   E6POS P2_G_1_App1Place={X 149.37352,Y -2.09811,Z 1001.61812,A -90,B 0,C 180,S 2,T 51,E1 0,E2 0,E3 0,E4 0,E5 0,E6 0}
   E6POS P2_G_1_App2Place={X 149.37352,Y -2.09821,Z 851.61778,A -90,B 0,C 180,S 2,T 51,E1 0,E2 0,E3 0,E4 0,E5 0,E6 0}
   E6POS P2_G_1_Place={X 49.37367,Y -2.09846,Z 651.61785,A -90,B 0,C 180,S 2,T 51,E1 0,E2 0,E3 0,E4 0,E5 0,E6 0}
   E6POS P2_G_2_App1Place={X 353.37436,Y 585.90188,Z 1001.61812,A -90,B 0,C 180,S 2,T 3,E1 0,E2 0,E3 0,E4 0,E5 0,E6 0}
   E6POS P2_G_2_App2Place={X 353.37434,Y 585.90171,Z 851.61778,A -90,B 0,C 180,S 2,T 3,E1 0,E2 0,E3 0,E4 0,E5 0,E6 0}
   E6POS P2_G_2_Place={X 253.37397,Y 585.90191,Z 651.61785,A -90,B 0,C 180,S 2,T 3,E1 0,E2 0,E3 0,E4 0,E5 0,E6 0}
   E6POS P2_G_3_App1Place={X 162.41236,Y 1308.69058,Z 1001.61812,A -90,B 0,C 180,S 2,T 35,E1 0,E2 0,E3 0,E4 0,E5 0,E6 0}
   E6POS P2_G_3_App2Place={X 162.41236,Y 1308.69069,Z 851.61778,A -90,B 0,C 180,S 2,T 35,E1 0,E2 0,E3 0,E4 0,E5 0,E6 0}
   E6POS P2_G_3_Place={X 49.37239,Y 1173.90187,Z 651.61785,A -90,B 0,C 180,S 2,T 35,E1 0,E2 0,E3 0,E4 0,E5 0,E6 0}
   E6POS P2_G_4_App1Place={X 559.12222,Y -2.23499,Z 1001.61812,A -90,B 0,C -180,S 2,T 19,E1 0,E2 0,E3 0,E4 0,E5 0,E6 0}
   E6POS P2_G_4_App2Place={X 559.12222,Y -2.235,Z 851.61778,A -90,B 0,C 180,S 2,T 19,E1 0,E2 0,E3 0,E4 0,E5 0,E6 0}
   E6POS P2_G_4_Place={X 457.3734,Y -26.09812,Z 651.61785,A -90,B 0,C 180,S 2,T 19,E1 0,E2 0,E3 0,E4 0,E5 0,E6 0}
   E6POS P2_G_5_App1Place={X 566.4018,Y 1306.30275,Z 1001.61812,A -90,B 0,C -180,S 2,T 3,E1 0,E2 0,E3 0,E4 0,E5 0,E6 0}
   E6POS P2_G_5_App2Place={X 566.4018,Y 1306.30279,Z 851.61778,A -90,B 0,C 180,S 2,T 3,E1 0,E2 0,E3 0,E4 0,E5 0,E6 0}
   E6POS P2_G_5_Place={X 343.37167,Y 1197.90666,Z 651.61785,A -90,B 0,C 180,S 2,T 3,E1 0,E2 0,E3 0,E4 0,E5 0,E6 0}
   E6POS P2_G_6_App1Place={X 770.4018,Y 1306.30275,Z 1001.61812,A -90,B 0,C -180,S 2,T 3,E1 0,E2 0,E3 0,E4 0,E5 0,E6 0}
   E6POS P2_G_6_App2Place={X 770.4018,Y 1306.30279,Z 851.61778,A -90,B 0,C 180,S 2,T 3,E1 0,E2 0,E3 0,E4 0,E5 0,E6 0}
   E6POS P2_G_6_Place={X 547.37167,Y 1197.90666,Z 651.61785,A -90,B 0,C 180,S 2,T 3,E1 0,E2 0,E3 0,E4 0,E5 0,E6 0}
   E6POS P2_G_7_App1Place={X 853.12026,Y 609.77279,Z 1001.61812,A -89.99997,B 0,C -180,S 2,T 3,E1 0,E2 0,E3 0,E4 0,E5 0,E6 0}
   E6POS P2_G_7_App2Place={X 853.12035,Y 609.77308,Z 851.61778,A -89.99997,B 0,C 180,S 2,T 3,E1 0,E2 0,E3 0,E4 0,E5 0,E6 0}
   E6POS P2_G_7_Place={X 751.37887,Y 612.61574,Z 651.61785,A -89.99997,B 0,C 180,S 2,T 3,E1 0,E2 0,E3 0,E4 0,E5 0,E6 0}
   E6POS P2_G_8_App1Place={X 753.12073,Y 609.77254,Z 1001.61812,A -90,B 0,C 180,S 2,T 3,E1 0,E2 0,E3 0,E4 0,E5 0,E6 0}
   E6POS P2_G_8_App2Place={X 753.12006,Y 654.77255,Z 851.61778,A -89.99997,B 0,C 180,S 2,T 3,E1 0,E2 0,E3 0,E4 0,E5 0,E6 0}
   E6POS P2_G_8_Place={X 753.12003,Y 654.77244,Z 651.61785,A -89.99997,B 0,C 180,S 2,T 3,E1 0,E2 0,E3 0,E4 0,E5 0,E6 0}
   E6POS P2_G_9_App1Place={X 753.12006,Y 654.77255,Z 1001.61812,A -89.99997,B 0,C 180,S 2,T 3,E1 0,E2 0,E3 0,E4 0,E5 0,E6 0}
   E6POS P2_G_9_App2Place={X 753.12053,Y 699.77216,Z 851.61778,A -90,B 0,C 180,S 2,T 3,E1 0,E2 0,E3 0,E4 0,E5 0,E6 0}
   E6POS P2_G_9_Place={X 753.12063,Y 699.77251,Z 651.61785,A -90,B 0,C 180,S 2,T 3,E1 0,E2 0,E3 0,E4 0,E5 0,E6 0}
   E6POS P2_G_10_App1Place={X 753.12053,Y 699.77216,Z 1001.61812,A -90,B 0,C 180,S 2,T 3,E1 0,E2 0,E3 0,E4 0,E5 0,E6 0}
   E6POS P2_G_10_App2Place={X 753.12058,Y 744.7725,Z 851.61778,A -90,B 0,C 180,S 2,T 3,E1 0,E2 0,E3 0,E4 0,E5 0,E6 0}
   E6POS P2_G_10_Place={X 753.12059,Y 744.77255,Z 651.61785,A -90,B 0,C 180,S 2,T 3,E1 0,E2 0,E3 0,E4 0,E5 0,E6 0}
   E6POS P2_G_11_App1Place={X 753.12058,Y 744.7725,Z 1001.61812,A -90,B 0,C 180,S 2,T 3,E1 0,E2 0,E3 0,E4 0,E5 0,E6 0}
   E6POS P2_G_11_App2Place={X 753.12054,Y 789.7722,Z 851.61778,A -90,B 0,C 180,S 2,T 3,E1 0,E2 0,E3 0,E4 0,E5 0,E6 0}
   E6POS P2_G_11_Place={X 753.12064,Y 789.7726,Z 651.61785,A -90,B 0,C 180,S 2,T 3,E1 0,E2 0,E3 0,E4 0,E5 0,E6 0}
   E6POS P2_G_12_App1Place={X 443.37199,Y 585.90705,Z 1001.61812,A -90,B 0,C -180,S 2,T 3,E1 0,E2 0,E3 0,E4 0,E5 0,E6 0}
   E6POS P2_G_12_App2Place={X 443.37195,Y 585.90667,Z 851.61778,A -90,B 0,C 180,S 2,T 3,E1 0,E2 0,E3 0,E4 0,E5 0,E6 0}
   E6POS P2_G_12_Place={X 343.37181,Y 585.90688,Z 651.61785,A -90,B 0,C 180,S 2,T 3,E1 0,E2 0,E3 0,E4 0,E5 0,E6 0}
   E6POS P2_G_13_App1Place={X 647.37185,Y -2.09309,Z 1001.61812,A -90,B 0,C -180,S 2,T 3,E1 0,E2 0,E3 0,E4 0,E5 0,E6 0}
   E6POS P2_G_13_App2Place={X 647.37173,Y -2.09348,Z 851.61778,A -90,B 0,C 180,S 2,T 3,E1 0,E2 0,E3 0,E4 0,E5 0,E6 0}
   E6POS P2_G_13_Place={X 547.37181,Y -2.0932,Z 651.61785,A -90,B 0,C 180,S 2,T 19,E1 0,E2 0,E3 0,E4 0,E5 0,E6 0}
   E6POS P2_G_14_App1Place={X 393.37089,Y 1223.90695,Z 1001.61812,A -90,B 0,C 180,S 2,T 3,E1 0,E2 0,E3 0,E4 0,E5 0,E6 0}
   E6POS P2_G_14_App2Place={X 393.37089,Y 1223.90695,Z 851.61778,A -90,B 0,C 180,S 2,T 3,E1 0,E2 0,E3 0,E4 0,E5 0,E6 0}
   E6POS P2_G_14_Place={X 343.37089,Y 1173.90695,Z 651.61785,A -90,B 0,C 180,S 2,T 3,E1 0,E2 0,E3 0,E4 0,E5 0,E6 0}
   E6POS P2_G_15_App1Place={X 853.11933,Y -26.09364,Z 1001.61812,A -90,B 0,C -180,S 2,T 3,E1 0,E2 0,E3 0,E4 0,E5 0,E6 0}
   E6POS P2_G_15_App2Place={X 853.11941,Y -26.09348,Z 851.61778,A -90,B 0,C 180,S 2,T 3,E1 0,E2 0,E3 0,E4 0,E5 0,E6 0}
   E6POS P2_G_15_Place={X 751.37143,Y -26.09385,Z 651.61785,A -90,B 0,C 180,S 2,T 19,E1 0,E2 0,E3 0,E4 0,E5 0,E6 0}
   E6POS P2_G_16_App1Place={X 737.36387,Y 1297.90653,Z 1001.61812,A -90,B 0,C -180,S 2,T 3,E1 0,E2 0,E3 0,E4 0,E5 0,E6 0}
   E6POS P2_G_16_App2Place={X 737.36384,Y 1297.90637,Z 851.61778,A -90,B 0,C 180,S 2,T 3,E1 0,E2 0,E3 0,E4 0,E5 0,E6 0}
   E6POS P2_G_16_Place={X 637.37555,Y 1197.90665,Z 651.61785,A -90,B 0,C 180,S 2,T 3,E1 0,E2 0,E3 0,E4 0,E5 0,E6 0}
   E6POS P2_G_17_App1Place={X 941.36387,Y 1297.90653,Z 1001.61812,A -90,B 0,C -180,S 2,T 3,E1 0,E2 0,E3 0,E4 0,E5 0,E6 0}
   E6POS P2_G_17_App2Place={X 941.36384,Y 1297.90637,Z 851.61778,A -90,B 0,C -180,S 2,T 3,E1 0,E2 0,E3 0,E4 0,E5 0,E6 0}
   E6POS P2_G_17_Place={X 841.37555,Y 1197.90665,Z 651.61785,A -90,B 0,C -180,S 2,T 3,E1 0,E2 0,E3 0,E4 0,E5 0,E6 0}
   E6POS P2_G_18_App1Place={X 75.37306,Y 583.87483,Z 1001.61812,A 90,B 0,C -180,S 2,T 35,E1 0,E2 0,E3 0,E4 0,E5 0,E6 0}
   E6POS P2_G_18_App2Place={X 75.37307,Y 583.87481,Z 851.61778,A 90,B 0,C 180,S 2,T 35,E1 0,E2 0,E3 0,E4 0,E5 0,E6 0}
   E6POS P2_G_18_Place={X 220.62117,Y 583.87476,Z 651.61785,A 90,B 0,C 180,S 2,T 35,E1 0,E2 0,E3 0,E4 0,E5 0,E6 0}
   E6POS P2_G_19_App1Place={X 220.62116,Y 583.87476,Z 1001.61812,A 90,B 0,C 180,S 2,T 35,E1 0,E2 0,E3 0,E4 0,E5 0,E6 0}
   E6POS P2_G_19_App2Place={X 220.62116,Y 538.87476,Z 851.61778,A 90,B 0,C 180,S 2,T 35,E1 0,E2 0,E3 0,E4 0,E5 0,E6 0}
   E6POS P2_G_19_Place={X 220.62116,Y 538.87476,Z 651.61785,A 90,B 0,C 180,S 2,T 35,E1 0,E2 0,E3 0,E4 0,E5 0,E6 0}
   E6POS P2_G_20_App1Place={X 220.62116,Y 538.87476,Z 1001.61812,A 90,B 0,C 180,S 2,T 35,E1 0,E2 0,E3 0,E4 0,E5 0,E6 0}
   E6POS P2_G_20_App2Place={X 220.62116,Y 493.87476,Z 851.61778,A 90,B 0,C 180,S 2,T 35,E1 0,E2 0,E3 0,E4 0,E5 0,E6 0}
   E6POS P2_G_20_Place={X 220.62116,Y 493.87476,Z 651.61785,A 90,B 0,C 180,S 2,T 35,E1 0,E2 0,E3 0,E4 0,E5 0,E6 0}
   E6POS P2_G_21_App1Place={X 220.62116,Y 493.87476,Z 1001.61812,A 90,B 0,C 180,S 2,T 35,E1 0,E2 0,E3 0,E4 0,E5 0,E6 0}
   E6POS P2_G_21_App2Place={X 220.62116,Y 448.87476,Z 851.61778,A 90,B 0,C 180,S 2,T 35,E1 0,E2 0,E3 0,E4 0,E5 0,E6 0}
   E6POS P2_G_21_Place={X 220.62116,Y 448.87476,Z 651.61785,A 90,B 0,C 180,S 2,T 35,E1 0,E2 0,E3 0,E4 0,E5 0,E6 0}
   E6POS P2_G_22_App1Place={X 220.62116,Y 448.87476,Z 1001.61812,A 90,B 0,C 180,S 2,T 35,E1 0,E2 0,E3 0,E4 0,E5 0,E6 0}
   E6POS P2_G_22_App2Place={X 220.62116,Y 403.87476,Z 851.61778,A 90,B 0,C 180,S 2,T 35,E1 0,E2 0,E3 0,E4 0,E5 0,E6 0}
   E6POS P2_G_22_Place={X 220.62116,Y 403.87476,Z 651.61785,A 90,B 0,C 180,S 2,T 35,E1 0,E2 0,E3 0,E4 0,E5 0,E6 0}

   ;ENDFOLD
   ;FOLD  MosaicoI_Pallet2

   E6POS P2_I_1_App1Place={X 246.53077,Y 662.7024,Z 986.30178,A -90,B 0,C 180,S 2,T 3,E1 0,E2 0,E3 0,E4 0,E5 0,E6 0}
   E6POS P2_I_1_App2Place={X 246.53091,Y 662.7025,Z 836.30179,A -90,B 0,C 180,S 2,T 3,E1 0,E2 0,E3 0,E4 0,E5 0,E6 0}
   E6POS P2_I_1_Place={X 120.2419,Y 563.31321,Z 652.09239,A -90,B 0,C 180,S 2,T 35,E1 0,E2 0,E3 0,E4 0,E5 0,E6 0}
   E6POS P2_I_2_App1Place={X 120.24188,Y 563.31279,Z 986.30178,A -90,B 0,C 180,S 2,T 35,E1 0,E2 0,E3 0,E4 0,E5 0,E6 0}
   E6POS P2_I_2_App2Place={X 120.24229,Y 624.31271,Z 836.30179,A -90,B 0,C 180,S 2,T 35,E1 0,E2 0,E3 0,E4 0,E5 0,E6 0}
   E6POS P2_I_2_Place={X 120.24227,Y 624.3123,Z 652.09239,A -90,B 0,C 180,S 2,T 35,E1 0,E2 0,E3 0,E4 0,E5 0,E6 0}
   E6POS P2_I_3_App1Place={X 120.24229,Y 624.31271,Z 986.30178,A -90,B 0,C 180,S 2,T 35,E1 0,E2 0,E3 0,E4 0,E5 0,E6 0}
   E6POS P2_I_3_App2Place={X 120.24194,Y 685.31244,Z 836.30179,A -90,B 0,C 180,S 2,T 35,E1 0,E2 0,E3 0,E4 0,E5 0,E6 0}
   E6POS P2_I_3_Place={X 120.24196,Y 685.31272,Z 652.09239,A -90,B 0,C 180,S 2,T 35,E1 0,E2 0,E3 0,E4 0,E5 0,E6 0}
   E6POS P2_I_4_App1Place={X 584.7347,Y 593.50005,Z 986.30178,A 90,B 0,C 180,S 2,T 35,E1 0,E2 0,E3 0,E4 0,E5 0,E6 0}
   E6POS P2_I_4_App2Place={X 584.73528,Y 593.49987,Z 836.30179,A 90,B 0,C 180,S 2,T 35,E1 0,E2 0,E3 0,E4 0,E5 0,E6 0}
   E6POS P2_I_4_Place={X 484.73518,Y 593.50008,Z 652.09239,A 90,B 0,C 180,S 2,T 35,E1 0,E2 0,E3 0,E4 0,E5 0,E6 0}
   E6POS P2_I_5_App1Place={X 942.73548,Y 593.50065,Z 986.30178,A 90,B 0,C 180,S 2,T 35,E1 0,E2 0,E3 0,E4 0,E5 0,E6 0}
   E6POS P2_I_5_App2Place={X 942.73575,Y 593.50015,Z 836.30179,A 90,B 0,C 180,S 2,T 35,E1 0,E2 0,E3 0,E4 0,E5 0,E6 0}
   E6POS P2_I_5_Place={X 842.73579,Y 593.50005,Z 652.09239,A 90,B 0,C 180,S 2,T 35,E1 0,E2 0,E3 0,E4 0,E5 0,E6 0}
   E6POS P2_I_6_App1Place={X 413.73426,Y 594.42093,Z 986.30178,A 90,B 0,C 180,S 2,T 35,E1 0,E2 0,E3 0,E4 0,E5 0,E6 0}
   E6POS P2_I_6_App2Place={X 413.73463,Y 594.42083,Z 836.30179,A 90,B 0,C 180,S 2,T 35,E1 0,E2 0,E3 0,E4 0,E5 0,E6 0}
   E6POS P2_I_6_Place={X 313.73464,Y 594.42082,Z 652.09239,A 90,B 0,C 180,S 2,T 35,E1 0,E2 0,E3 0,E4 0,E5 0,E6 0}
   E6POS P2_I_7_App1Place={X 771.7338,Y 594.4204,Z 986.30178,A 90,B 0,C 180,S 2,T 35,E1 0,E2 0,E3 0,E4 0,E5 0,E6 0}
   E6POS P2_I_7_App2Place={X 771.73418,Y 594.4208,Z 836.30179,A 90,B 0,C 180,S 2,T 35,E1 0,E2 0,E3 0,E4 0,E5 0,E6 0}
   E6POS P2_I_7_Place={X 671.73443,Y 594.42068,Z 652.09239,A 90,B 0,C 180,S 2,T 35,E1 0,E2 0,E3 0,E4 0,E5 0,E6 0}
   E6POS P2_I_8_App1Place={X 936.24205,Y 563.31282,Z 986.30178,A -90,B 0,C 180,S 2,T 3,E1 0,E2 0,E3 0,E4 0,E5 0,E6 0}
   E6POS P2_I_8_App2Place={X 936.24164,Y 563.31281,Z 836.30179,A -90,B 0,C 180,S 2,T 3,E1 0,E2 0,E3 0,E4 0,E5 0,E6 0}
   E6POS P2_I_8_Place={X 836.24218,Y 563.31266,Z 652.09239,A -90,B 0,C 180,S 2,T 3,E1 0,E2 0,E3 0,E4 0,E5 0,E6 0}
   E6POS P2_I_9_App1Place={X 836.24219,Y 563.31262,Z 986.30178,A -90,B 0,C 180,S 2,T 3,E1 0,E2 0,E3 0,E4 0,E5 0,E6 0}
   E6POS P2_I_9_App2Place={X 836.24173,Y 624.31272,Z 836.30179,A -90,B 0,C 180,S 2,T 3,E1 0,E2 0,E3 0,E4 0,E5 0,E6 0}
   E6POS P2_I_9_Place={X 836.24181,Y 624.31245,Z 652.09239,A -90,B 0,C 180,S 2,T 3,E1 0,E2 0,E3 0,E4 0,E5 0,E6 0}
   E6POS P2_I_10_App1Place={X 836.24173,Y 624.31272,Z 986.30178,A -90,B 0,C 180,S 2,T 3,E1 0,E2 0,E3 0,E4 0,E5 0,E6 0}
   E6POS P2_I_10_App2Place={X 836.24228,Y 685.31292,Z 836.30179,A -90,B 0,C 180,S 2,T 3,E1 0,E2 0,E3 0,E4 0,E5 0,E6 0}
   E6POS P2_I_10_Place={X 836.24232,Y 685.3128,Z 652.09239,A -90,B 0,C 180,S 2,T 3,E1 0,E2 0,E3 0,E4 0,E5 0,E6 0}

   ;ENDFOLD
   ;FOLD  MosaicoJ_Pallet2

   E6POS P2_J_1_App1Place={X 205.12202,Y 673.01054,Z 986.30252,A 90,B 0,C 180,S 2,T 35,E1 0,E2 0,E3 0,E4 0,E5 0,E6 0}
   E6POS P2_J_1_App2Place={X 205.12222,Y 673.01047,Z 786.30223,A 90,B 0,C 180,S 2,T 35,E1 0,E2 0,E3 0,E4 0,E5 0,E6 0}
   E6POS P2_J_1_Place={X 83.2071,Y 563.55362,Z 666.3006,A 90,B 0,C 180,S 2,T 35,E1 0,E2 0,E3 0,E4 0,E5 0,E6 0}
   E6POS P2_J_2_App1Place={X 996.70818,Y 190.44821,Z 986.30252,A -180,B 0,C -180,S 2,T 35,E1 0,E2 0,E3 0,E4 0,E5 0,E6 0}
   E6POS P2_J_2_App2Place={X 996.70793,Y 190.44835,Z 786.30223,A -180,B 0,C 180,S 2,T 35,E1 0,E2 0,E3 0,E4 0,E5 0,E6 0}
   E6POS P2_J_2_Place={X 896.70882,Y 90.44837,Z 666.3006,A -180,B 0,C -180,S 2,T 51,E1 0,E2 0,E3 0,E4 0,E5 0,E6 0}
   E6POS P2_J_3_App1Place={X 996.70874,Y 479.44951,Z 986.30252,A -180,B 0,C 180,S 2,T 35,E1 0,E2 0,E3 0,E4 0,E5 0,E6 0}
   E6POS P2_J_3_App2Place={X 996.70888,Y 479.44931,Z 786.30223,A -180,B 0,C 180,S 2,T 35,E1 0,E2 0,E3 0,E4 0,E5 0,E6 0}
   E6POS P2_J_3_Place={X 896.7079,Y 379.44856,Z 666.3006,A -180,B 0,C 180,S 2,T 35,E1 0,E2 0,E3 0,E4 0,E5 0,E6 0}
   E6POS P2_J_4_App1Place={X 996.70922,Y 768.44904,Z 986.30252,A -180,B 0,C 180,S 2,T 35,E1 0,E2 0,E3 0,E4 0,E5 0,E6 0}
   E6POS P2_J_4_App2Place={X 996.70882,Y 768.44907,Z 786.30223,A -180,B 0,C 180,S 2,T 35,E1 0,E2 0,E3 0,E4 0,E5 0,E6 0}
   E6POS P2_J_4_Place={X 896.708,Y 668.44849,Z 666.3006,A -180,B 0,C 180,S 2,T 35,E1 0,E2 0,E3 0,E4 0,E5 0,E6 0}
   E6POS P2_J_5_App1Place={X 996.70917,Y 1057.44893,Z 986.30252,A -180,B 0,C 180,S 2,T 35,E1 0,E2 0,E3 0,E4 0,E5 0,E6 0}
   E6POS P2_J_5_App2Place={X 996.70891,Y 1057.44895,Z 786.30223,A -180,B 0,C -180,S 2,T 35,E1 0,E2 0,E3 0,E4 0,E5 0,E6 0}
   E6POS P2_J_5_Place={X 896.7083,Y 957.44855,Z 666.3006,A -180,B 0,C 180,S 2,T 35,E1 0,E2 0,E3 0,E4 0,E5 0,E6 0}
   E6POS P2_J_6_App1Place={X 624.70927,Y 190.44867,Z 986.30252,A -180,B 0,C 180,S 2,T 35,E1 0,E2 0,E3 0,E4 0,E5 0,E6 0}
   E6POS P2_J_6_App2Place={X 624.70884,Y 190.44885,Z 786.30223,A -180,B 0,C -180,S 2,T 35,E1 0,E2 0,E3 0,E4 0,E5 0,E6 0}
   E6POS P2_J_6_Place={X 624.70888,Y 90.44835,Z 666.3006,A -180,B 0,C 180,S 2,T 35,E1 0,E2 0,E3 0,E4 0,E5 0,E6 0}
   E6POS P2_J_7_App1Place={X 624.70769,Y 479.44883,Z 986.30252,A -180,B 0,C 180,S 2,T 35,E1 0,E2 0,E3 0,E4 0,E5 0,E6 0}
   E6POS P2_J_7_App2Place={X 624.70799,Y 479.4485,Z 786.30223,A -180,B 0,C 180,S 2,T 35,E1 0,E2 0,E3 0,E4 0,E5 0,E6 0}
   E6POS P2_J_7_Place={X 624.70786,Y 379.44821,Z 666.3006,A -180,B 0,C -180,S 2,T 35,E1 0,E2 0,E3 0,E4 0,E5 0,E6 0}
   E6POS P2_J_8_App1Place={X 624.70801,Y 768.44835,Z 986.30252,A -180,B 0,C 180,S 2,T 35,E1 0,E2 0,E3 0,E4 0,E5 0,E6 0}
   E6POS P2_J_8_App2Place={X 624.70825,Y 768.44844,Z 786.30223,A -180,B 0,C 180,S 2,T 35,E1 0,E2 0,E3 0,E4 0,E5 0,E6 0}
   E6POS P2_J_8_Place={X 624.70846,Y 668.44829,Z 666.3006,A -180,B 0,C -180,S 2,T 35,E1 0,E2 0,E3 0,E4 0,E5 0,E6 0}
   E6POS P2_J_9_App1Place={X 624.70855,Y 1057.44886,Z 986.30252,A -180,B 0,C -180,S 2,T 35,E1 0,E2 0,E3 0,E4 0,E5 0,E6 0}
   E6POS P2_J_9_App2Place={X 624.70849,Y 1057.44878,Z 786.30223,A -180,B 0,C -180,S 2,T 35,E1 0,E2 0,E3 0,E4 0,E5 0,E6 0}
   E6POS P2_J_9_Place={X 624.7086,Y 957.44847,Z 666.3006,A -180,B 0,C 180,S 2,T 35,E1 0,E2 0,E3 0,E4 0,E5 0,E6 0}
   E6POS P2_J_10_App1Place={X 867.21049,Y 562.58511,Z 986.30252,A 90,B 0,C 180,S 2,T 35,E1 0,E2 0,E3 0,E4 0,E5 0,E6 0}
   E6POS P2_J_10_App2Place={X 867.21029,Y 562.58552,Z 786.30223,A 90,B 0,C 180,S 2,T 35,E1 0,E2 0,E3 0,E4 0,E5 0,E6 0}
   E6POS P2_J_10_Place={X 767.21058,Y 562.5858,Z 666.3006,A 90,B 0,C 180,S 2,T 35,E1 0,E2 0,E3 0,E4 0,E5 0,E6 0}

   ;ENDFOLD
   ;FOLD  MosaicoK_Pallet2

   E6POS P2_K_1_App1Place={X 965.18951,Y 160.47376,Z 1002.77257,A -180,B 0,C 180,S 2,T 35,E1 0,E2 0,E3 0,E4 0,E5 0,E6 0}
   E6POS P2_K_1_App2Place={X 965.18946,Y 160.47317,Z 802.77226,A -180,B 0,C 180,S 2,T 35,E1 0,E2 0,E3 0,E4 0,E5 0,E6 0}
   E6POS P2_K_1_Place={X 965.18981,Y 60.47307,Z 652.77183,A -180,B 0,C -180,S 2,T 51,E1 0,E2 0,E3 0,E4 0,E5 0,E6 0}
   E6POS P2_K_2_App1Place={X 289.34869,Y 416.70488,Z 1002.77257,A -180,B 0,C 180,S 2,T 35,E1 0,E2 0,E3 0,E4 0,E5 0,E6 0}
   E6POS P2_K_2_App2Place={X 289.34829,Y 416.70443,Z 802.77226,A -180,B 0,C -180,S 2,T 35,E1 0,E2 0,E3 0,E4 0,E5 0,E6 0}
   E6POS P2_K_2_Place={X 289.34787,Y 316.70418,Z 652.77183,A -180,B 0,C -180,S 2,T 51,E1 0,E2 0,E3 0,E4 0,E5 0,E6 0}
   E6POS P2_K_3_App1Place={X 709.18337,Y 836.49354,Z 1002.77257,A -180,B 0,C 180,S 2,T 35,E1 0,E2 0,E3 0,E4 0,E5 0,E6 0}
   E6POS P2_K_3_App2Place={X 709.18357,Y 836.4934,Z 802.77226,A -180,B 0,C 180,S 2,T 35,E1 0,E2 0,E3 0,E4 0,E5 0,E6 0}
   E6POS P2_K_3_Place={X 709.18379,Y 736.49338,Z 652.77183,A -180,B 0,C -180,S 2,T 35,E1 0,E2 0,E3 0,E4 0,E5 0,E6 0}
   E6POS P2_K_4_App1Place={X 33.34909,Y 1092.70494,Z 1002.77257,A -180,B 0,C -180,S 2,T 35,E1 0,E2 0,E3 0,E4 0,E5 0,E6 0}
   E6POS P2_K_4_App2Place={X 33.34872,Y 1092.70456,Z 802.77226,A -180,B 0,C -180,S 2,T 35,E1 0,E2 0,E3 0,E4 0,E5 0,E6 0}
   E6POS P2_K_4_Place={X 33.34906,Y 992.70434,Z 652.77183,A -180,B 0,C 180,S 2,T 35,E1 0,E2 0,E3 0,E4 0,E5 0,E6 0}
   E6POS P2_K_5_App1Place={X 135.86643,Y -91.91437,Z 1002.77257,A 90,B 0,C 180,S 2,T 51,E1 0,E2 0,E3 0,E4 0,E5 0,E6 0}
   E6POS P2_K_5_App2Place={X 135.86633,Y -91.91463,Z 802.77226,A 90,B 0,C 180,S 2,T 51,E1 0,E2 0,E3 0,E4 0,E5 0,E6 0}
   E6POS P2_K_5_Place={X 230.11027,Y 4.30843,Z 652.77183,A 90,B 0,C 180,S 2,T 51,E1 0,E2 0,E3 0,E4 0,E5 0,E6 0}
   E6POS P2_K_6_App1Place={X 867.49583,Y 1243.09331,Z 1002.77257,A -90.00003,B 0,C 180,S 2,T 3,E1 0,E2 0,E3 0,E4 0,E5 0,E6 0}
   E6POS P2_K_6_App2Place={X 867.4955,Y 1243.0937,Z 802.77226,A -90.00001,B 0,C 180,S 2,T 3,E1 0,E2 0,E3 0,E4 0,E5 0,E6 0}
   E6POS P2_K_6_Place={X 767.4955,Y 1193.0937,Z 652.77183,A -90.00001,B 0,C 180,S 2,T 3,E1 0,E2 0,E3 0,E4 0,E5 0,E6 0}
   E6POS P2_K_7_App1Place={X 709.18372,Y 160.49371,Z 1002.77257,A -180,B 0,C 180,S 2,T 35,E1 0,E2 0,E3 0,E4 0,E5 0,E6 0}
   E6POS P2_K_7_App2Place={X 709.18356,Y 160.49366,Z 802.77226,A -180,B 0,C 180,S 2,T 35,E1 0,E2 0,E3 0,E4 0,E5 0,E6 0}
   E6POS P2_K_7_Place={X 709.18265,Y 60.49314,Z 652.77183,A -180,B 0,C 180,S 2,T 35,E1 0,E2 0,E3 0,E4 0,E5 0,E6 0}
   E6POS P2_K_8_App1Place={X 33.34874,Y 416.70446,Z 1002.77257,A -180,B 0,C 180,S 2,T 35,E1 0,E2 0,E3 0,E4 0,E5 0,E6 0}
   E6POS P2_K_8_App2Place={X 33.34863,Y 416.70468,Z 802.77226,A -180,B 0,C -180,S 2,T 35,E1 0,E2 0,E3 0,E4 0,E5 0,E6 0}
   E6POS P2_K_8_Place={X 33.3492,Y 316.7046,Z 652.77183,A -180,B 0,C -180,S 2,T 35,E1 0,E2 0,E3 0,E4 0,E5 0,E6 0}
   E6POS P2_K_9_App1Place={X 965.18407,Y 836.49236,Z 1002.77257,A -180,B 0,C 180,S 2,T 35,E1 0,E2 0,E3 0,E4 0,E5 0,E6 0}
   E6POS P2_K_9_App2Place={X 965.18406,Y 836.49238,Z 802.77226,A -180,B 0,C 180,S 2,T 35,E1 0,E2 0,E3 0,E4 0,E5 0,E6 0}
   E6POS P2_K_9_Place={X 965.18419,Y 736.49329,Z 652.77183,A -180,B 0,C 180,S 2,T 35,E1 0,E2 0,E3 0,E4 0,E5 0,E6 0}
   E6POS P2_K_10_App1Place={X 289.34853,Y 1092.70485,Z 1002.77257,A -180,B 0,C 180,S 2,T 35,E1 0,E2 0,E3 0,E4 0,E5 0,E6 0}
   E6POS P2_K_10_App2Place={X 289.34898,Y 1092.70437,Z 802.77226,A -180,B 0,C 180,S 2,T 35,E1 0,E2 0,E3 0,E4 0,E5 0,E6 0}
   E6POS P2_K_10_Place={X 289.34887,Y 992.70441,Z 652.77183,A -180,B 0,C -180,S 2,T 35,E1 0,E2 0,E3 0,E4 0,E5 0,E6 0}
   E6POS P2_K_11_App1Place={X 132.98721,Y 1243.0855,Z 1002.77257,A -90,B 0,C 180,S 2,T 35,E1 0,E2 0,E3 0,E4 0,E5 0,E6 0}
   E6POS P2_K_11_App2Place={X 132.98733,Y 1243.08625,Z 802.77226,A -90,B 0,C 180,S 2,T 35,E1 0,E2 0,E3 0,E4 0,E5 0,E6 0}
   E6POS P2_K_11_Place={X 232.98733,Y 1193.08625,Z 652.77183,A -90,B 0,C 180,S 2,T 3,E1 0,E2 0,E3 0,E4 0,E5 0,E6 0}
   E6POS P2_K_12_App1Place={X 864.59574,Y -45.68689,Z 1002.77257,A 90,B 0,C 180,S 2,T 35,E1 0,E2 0,E3 0,E4 0,E5 0,E6 0}
   E6POS P2_K_12_App2Place={X 864.59587,Y -45.68653,Z 802.77226,A 90,B 0,C 180,S 2,T 35,E1 0,E2 0,E3 0,E4 0,E5 0,E6 0}
   E6POS P2_K_12_Place={X 764.59587,Y 4.31347,Z 652.77183,A 90,B 0,C 180,S 2,T 51,E1 0,E2 0,E3 0,E4 0,E5 0,E6 0}

   ;ENDFOLD
   ;FOLD  MosaicoL_Pallet2

   E6POS P2_L_1_App1Place={X 168.06418,Y 598.29338,Z 1070.17203,A -89.99997,B 0,C -180,S 2,T 35,E1 0,E2 0,E3 0,E4 0,E5 0,E6 0}
   E6POS P2_L_1_App2Place={X 168.06418,Y 598.29353,Z 870.17216,A -89.99997,B 0,C 180,S 2,T 35,E1 0,E2 0,E3 0,E4 0,E5 0,E6 0}
   E6POS P2_L_1_Place={X 68.06526,Y 598.29341,Z 670.17152,A -90,B 0,C 180,S 2,T 35,E1 0,E2 0,E3 0,E4 0,E5 0,E6 0}
   E6POS P2_L_2_App1Place={X 432.06392,Y 598.29328,Z 1070.17203,A -89.99997,B 0,C -180,S 2,T 3,E1 0,E2 0,E3 0,E4 0,E5 0,E6 0}
   E6POS P2_L_2_App2Place={X 432.06389,Y 598.29299,Z 870.17216,A -89.99997,B 0,C 180,S 2,T 3,E1 0,E2 0,E3 0,E4 0,E5 0,E6 0}
   E6POS P2_L_2_Place={X 332.06426,Y 598.2932,Z 670.17152,A -89.99997,B 0,C 180,S 2,T 3,E1 0,E2 0,E3 0,E4 0,E5 0,E6 0}
   E6POS P2_L_3_App1Place={X 696.09642,Y 672.2385,Z 1070.17203,A -90,B 0,C -180,S 2,T 3,E1 0,E2 0,E3 0,E4 0,E5 0,E6 0}
   E6POS P2_L_3_App2Place={X 696.09645,Y 672.23864,Z 870.17216,A -90,B 0,C 180,S 2,T 3,E1 0,E2 0,E3 0,E4 0,E5 0,E6 0}
   E6POS P2_L_3_Place={X 596.09736,Y 672.23879,Z 670.17152,A -90,B 0,C 180,S 2,T 3,E1 0,E2 0,E3 0,E4 0,E5 0,E6 0}
   E6POS P2_L_4_App1Place={X 596.09735,Y 672.23874,Z 1070.17203,A -90,B 0,C 180,S 2,T 3,E1 0,E2 0,E3 0,E4 0,E5 0,E6 0}
   E6POS P2_L_4_App2Place={X 596.09692,Y 648.23875,Z 870.17216,A -90,B 0,C 180,S 2,T 3,E1 0,E2 0,E3 0,E4 0,E5 0,E6 0}
   E6POS P2_L_4_Place={X 596.09685,Y 648.23836,Z 670.17152,A -90,B 0,C 180,S 2,T 3,E1 0,E2 0,E3 0,E4 0,E5 0,E6 0}
   E6POS P2_L_5_App1Place={X 596.09692,Y 648.23875,Z 1070.17203,A -90,B 0,C 180,S 2,T 3,E1 0,E2 0,E3 0,E4 0,E5 0,E6 0}
   E6POS P2_L_5_App2Place={X 596.09676,Y 624.23876,Z 870.17216,A -90,B 0,C 180,S 2,T 3,E1 0,E2 0,E3 0,E4 0,E5 0,E6 0}
   E6POS P2_L_5_Place={X 596.09673,Y 624.23857,Z 670.17152,A -90,B 0,C 180,S 2,T 3,E1 0,E2 0,E3 0,E4 0,E5 0,E6 0}
   E6POS P2_L_6_App1Place={X 596.09676,Y 624.23876,Z 1070.17203,A -90,B 0,C 180,S 2,T 3,E1 0,E2 0,E3 0,E4 0,E5 0,E6 0}
   E6POS P2_L_6_App2Place={X 596.09655,Y 600.23828,Z 870.17216,A -90,B 0,C 180,S 2,T 3,E1 0,E2 0,E3 0,E4 0,E5 0,E6 0}
   E6POS P2_L_6_Place={X 596.09665,Y 600.23877,Z 670.17152,A -90,B 0,C 180,S 2,T 3,E1 0,E2 0,E3 0,E4 0,E5 0,E6 0}
   E6POS P2_L_7_App1Place={X 922.09632,Y 672.23843,Z 1070.17203,A -90,B 0,C -180,S 2,T 3,E1 0,E2 0,E3 0,E4 0,E5 0,E6 0}
   E6POS P2_L_7_App2Place={X 922.09645,Y 672.23879,Z 870.17216,A -90,B 0,C 180,S 2,T 3,E1 0,E2 0,E3 0,E4 0,E5 0,E6 0}
   E6POS P2_L_7_Place={X 822.09609,Y 672.23876,Z 670.17152,A -90,B 0,C 180,S 2,T 3,E1 0,E2 0,E3 0,E4 0,E5 0,E6 0}
   E6POS P2_L_8_App1Place={X 822.09616,Y 672.23897,Z 1070.17203,A -90,B 0,C 180,S 2,T 3,E1 0,E2 0,E3 0,E4 0,E5 0,E6 0}
   E6POS P2_L_8_App2Place={X 822.09694,Y 648.23821,Z 870.17216,A -90,B 0,C 180,S 2,T 3,E1 0,E2 0,E3 0,E4 0,E5 0,E6 0}
   E6POS P2_L_8_Place={X 822.0969,Y 648.23809,Z 670.17152,A -90,B 0,C 180,S 2,T 3,E1 0,E2 0,E3 0,E4 0,E5 0,E6 0}
   E6POS P2_L_9_App1Place={X 822.09694,Y 648.23821,Z 1070.17203,A -90,B 0,C 180,S 2,T 3,E1 0,E2 0,E3 0,E4 0,E5 0,E6 0}
   E6POS P2_L_9_App2Place={X 822.09613,Y 624.23895,Z 870.17216,A -90,B 0,C 180,S 2,T 3,E1 0,E2 0,E3 0,E4 0,E5 0,E6 0}
   E6POS P2_L_9_Place={X 822.09596,Y 624.23841,Z 670.17152,A -90,B 0,C 180,S 2,T 3,E1 0,E2 0,E3 0,E4 0,E5 0,E6 0}
   E6POS P2_L_10_App1Place={X 822.09613,Y 624.23895,Z 1070.17203,A -90,B 0,C 180,S 2,T 3,E1 0,E2 0,E3 0,E4 0,E5 0,E6 0}
   E6POS P2_L_10_App2Place={X 822.09631,Y 600.23873,Z 870.17216,A -90,B 0,C 180,S 2,T 3,E1 0,E2 0,E3 0,E4 0,E5 0,E6 0}
   E6POS P2_L_10_Place={X 822.09637,Y 600.23894,Z 670.17152,A -90,B 0,C 180,S 2,T 3,E1 0,E2 0,E3 0,E4 0,E5 0,E6 0}
   E6POS P2_L_11_App1Place={X 168.09611,Y 672.2385,Z 1070.17203,A -90,B 0,C 180,S 2,T 35,E1 0,E2 0,E3 0,E4 0,E5 0,E6 0}
   E6POS P2_L_11_App2Place={X 168.09611,Y 672.2387,Z 870.17216,A -90,B 0,C 180,S 2,T 35,E1 0,E2 0,E3 0,E4 0,E5 0,E6 0}
   E6POS P2_L_11_Place={X 68.09697,Y 672.23897,Z 670.17152,A -90,B 0,C 180,S 2,T 35,E1 0,E2 0,E3 0,E4 0,E5 0,E6 0}
   E6POS P2_L_12_App1Place={X 68.09697,Y 672.23896,Z 1070.17203,A -90,B 0,C 180,S 2,T 35,E1 0,E2 0,E3 0,E4 0,E5 0,E6 0}
   E6POS P2_L_12_App2Place={X 68.09599,Y 648.23858,Z 870.17216,A -90,B 0,C 180,S 2,T 35,E1 0,E2 0,E3 0,E4 0,E5 0,E6 0}
   E6POS P2_L_12_Place={X 68.09599,Y 648.23861,Z 670.17152,A -90,B 0,C 180,S 2,T 35,E1 0,E2 0,E3 0,E4 0,E5 0,E6 0}
   E6POS P2_L_13_App1Place={X 68.09599,Y 648.23858,Z 1070.17203,A -90,B 0,C 180,S 2,T 35,E1 0,E2 0,E3 0,E4 0,E5 0,E6 0}
   E6POS P2_L_13_App2Place={X 68.09686,Y 624.23871,Z 870.17216,A -90,B 0,C 180,S 2,T 35,E1 0,E2 0,E3 0,E4 0,E5 0,E6 0}
   E6POS P2_L_13_Place={X 68.09685,Y 624.23882,Z 670.17152,A -90,B 0,C 180,S 2,T 35,E1 0,E2 0,E3 0,E4 0,E5 0,E6 0}
   E6POS P2_L_14_App1Place={X 68.09686,Y 624.23871,Z 1070.17203,A -90,B 0,C 180,S 2,T 35,E1 0,E2 0,E3 0,E4 0,E5 0,E6 0}
   E6POS P2_L_14_App2Place={X 68.09658,Y 600.23864,Z 870.17216,A -90,B 0,C 180,S 2,T 35,E1 0,E2 0,E3 0,E4 0,E5 0,E6 0}
   E6POS P2_L_14_Place={X 68.09658,Y 600.2387,Z 670.17152,A -90,B 0,C 180,S 2,T 35,E1 0,E2 0,E3 0,E4 0,E5 0,E6 0}
   E6POS P2_L_15_App1Place={X 394.0962,Y 672.23855,Z 1070.17203,A -90,B 0,C -180,S 2,T 3,E1 0,E2 0,E3 0,E4 0,E5 0,E6 0}
   E6POS P2_L_15_App2Place={X 394.09624,Y 672.23892,Z 870.17216,A -90,B 0,C 180,S 2,T 3,E1 0,E2 0,E3 0,E4 0,E5 0,E6 0}
   E6POS P2_L_15_Place={X 294.09682,Y 672.23896,Z 670.17152,A -90,B 0,C 180,S 2,T 3,E1 0,E2 0,E3 0,E4 0,E5 0,E6 0}
   E6POS P2_L_16_App1Place={X 294.09682,Y 672.23888,Z 1070.17203,A -90,B 0,C 180,S 2,T 3,E1 0,E2 0,E3 0,E4 0,E5 0,E6 0}
   E6POS P2_L_16_App2Place={X 294.09703,Y 648.23826,Z 870.17216,A -90,B 0,C 180,S 2,T 3,E1 0,E2 0,E3 0,E4 0,E5 0,E6 0}
   E6POS P2_L_16_Place={X 294.09704,Y 648.23851,Z 670.17152,A -90,B 0,C 180,S 2,T 3,E1 0,E2 0,E3 0,E4 0,E5 0,E6 0}
   E6POS P2_L_17_App1Place={X 294.09703,Y 648.23826,Z 1070.17203,A -90,B 0,C 180,S 2,T 3,E1 0,E2 0,E3 0,E4 0,E5 0,E6 0}
   E6POS P2_L_17_App2Place={X 294.09602,Y 624.23846,Z 870.17216,A -90,B 0,C 180,S 2,T 3,E1 0,E2 0,E3 0,E4 0,E5 0,E6 0}
   E6POS P2_L_17_Place={X 294.09601,Y 624.23832,Z 670.17152,A -90,B 0,C 180,S 2,T 3,E1 0,E2 0,E3 0,E4 0,E5 0,E6 0}
   E6POS P2_L_18_App1Place={X 294.09602,Y 624.23846,Z 1070.17203,A -90,B 0,C 180,S 2,T 3,E1 0,E2 0,E3 0,E4 0,E5 0,E6 0}
   E6POS P2_L_18_App2Place={X 294.09608,Y 600.23829,Z 870.17216,A -90,B 0,C 180,S 2,T 3,E1 0,E2 0,E3 0,E4 0,E5 0,E6 0}
   E6POS P2_L_18_Place={X 294.0961,Y 600.23879,Z 670.17152,A -90,B 0,C 180,S 2,T 3,E1 0,E2 0,E3 0,E4 0,E5 0,E6 0}
   E6POS P2_L_19_App1Place={X 620.06432,Y 598.2933,Z 1070.17203,A -90,B 0,C -180,S 2,T 3,E1 0,E2 0,E3 0,E4 0,E5 0,E6 0}
   E6POS P2_L_19_App2Place={X 620.06428,Y 598.29308,Z 870.17216,A -90,B 0,C 180,S 2,T 3,E1 0,E2 0,E3 0,E4 0,E5 0,E6 0}
   E6POS P2_L_19_Place={X 520.06414,Y 598.29313,Z 670.17152,A -89.99997,B 0,C 180,S 2,T 3,E1 0,E2 0,E3 0,E4 0,E5 0,E6 0}
   E6POS P2_L_20_App1Place={X 884.0641,Y 598.29347,Z 1070.17203,A -89.99997,B 0,C 180,S 2,T 3,E1 0,E2 0,E3 0,E4 0,E5 0,E6 0}
   E6POS P2_L_20_App2Place={X 884.06402,Y 598.29325,Z 870.17216,A -89.99997,B 0,C 180,S 2,T 3,E1 0,E2 0,E3 0,E4 0,E5 0,E6 0}
   E6POS P2_L_20_Place={X 784.0648,Y 598.29314,Z 670.17152,A -90,B 0,C 180,S 2,T 3,E1 0,E2 0,E3 0,E4 0,E5 0,E6 0}

   ;ENDFOLD
   ;FOLD  MosaicoM_Pallet2

   E6POS P2_M_1_App1Place={X 185.75082,Y 502.65459,Z 990.17089,A -90,B 0,C 180,S 2,T 35,E1 0,E2 0,E3 0,E4 0,E5 0,E6 0}
   E6POS P2_M_1_App2Place={X 185.75082,Y 502.65481,Z 840.17071,A -90,B 0,C 180,S 2,T 35,E1 0,E2 0,E3 0,E4 0,E5 0,E6 0}
   E6POS P2_M_1_Place={X 60.91841,Y 601.45505,Z 670.17075,A -90,B 0,C 180,S 2,T 35,E1 0,E2 0,E3 0,E4 0,E5 0,E6 0}
   E6POS P2_M_2_App1Place={X 583.64026,Y 604.96255,Z 990.17089,A 90,B 0,C 180,S 2,T 35,E1 0,E2 0,E3 0,E4 0,E5 0,E6 0}
   E6POS P2_M_2_App2Place={X 583.64023,Y 604.96238,Z 840.17071,A 90,B 0,C 180,S 2,T 35,E1 0,E2 0,E3 0,E4 0,E5 0,E6 0}
   E6POS P2_M_2_Place={X 483.6401,Y 604.96221,Z 670.17075,A 90,B 0,C 180,S 2,T 35,E1 0,E2 0,E3 0,E4 0,E5 0,E6 0}
   E6POS P2_M_3_App1Place={X 969.64098,Y 604.96245,Z 990.17089,A 90,B 0,C 180,S 2,T 35,E1 0,E2 0,E3 0,E4 0,E5 0,E6 0}
   E6POS P2_M_3_App2Place={X 969.64086,Y 604.96213,Z 840.17071,A 90,B 0,C 180,S 2,T 35,E1 0,E2 0,E3 0,E4 0,E5 0,E6 0}
   E6POS P2_M_3_Place={X 869.64032,Y 604.96203,Z 670.17075,A 90,B 0,C 180,S 2,T 35,E1 0,E2 0,E3 0,E4 0,E5 0,E6 0}
   E6POS P2_M_4_App1Place={X 350.64914,Y 605.90332,Z 990.17089,A 90,B 0,C 180,S 2,T 35,E1 0,E2 0,E3 0,E4 0,E5 0,E6 0}
   E6POS P2_M_4_App2Place={X 350.64912,Y 605.90307,Z 840.17071,A 90,B 0,C 180,S 2,T 35,E1 0,E2 0,E3 0,E4 0,E5 0,E6 0}
   E6POS P2_M_4_Place={X 250.64929,Y 605.90345,Z 670.17075,A 90,B 0,C 180,S 2,T 35,E1 0,E2 0,E3 0,E4 0,E5 0,E6 0}
   E6POS P2_M_5_App1Place={X 736.64913,Y 605.90366,Z 990.17089,A 90,B 0,C 180,S 2,T 35,E1 0,E2 0,E3 0,E4 0,E5 0,E6 0}
   E6POS P2_M_5_App2Place={X 736.64908,Y 605.90347,Z 840.17071,A 90,B 0,C 180,S 2,T 35,E1 0,E2 0,E3 0,E4 0,E5 0,E6 0}
   E6POS P2_M_5_Place={X 636.64962,Y 605.90316,Z 670.17075,A 90,B 0,C 180,S 2,T 35,E1 0,E2 0,E3 0,E4 0,E5 0,E6 0}
   E6POS P2_M_6_App1Place={X 957.7513,Y 505.60753,Z 990.17089,A -90,B 0,C -180,S 2,T 3,E1 0,E2 0,E3 0,E4 0,E5 0,E6 0}
   E6POS P2_M_6_App2Place={X 957.75127,Y 505.60744,Z 840.17071,A -90,B 0,C -180,S 2,T 3,E1 0,E2 0,E3 0,E4 0,E5 0,E6 0}
   E6POS P2_M_6_Place={X 832.91967,Y 604.65501,Z 670.17075,A -90,B 0,C 180,S 2,T 3,E1 0,E2 0,E3 0,E4 0,E5 0,E6 0}

   ;ENDFOLD
   ;FOLD  MosaicoN_Pallet2

   E6POS P2_N_1_App1Place={X 133.08061,Y 567.70535,Z 953.39146,A 90,B 0,C 180,S 2,T 35,E1 0,E2 0,E3 0,E4 0,E5 0,E6 0}
   E6POS P2_N_1_App2Place={X 133.08067,Y 567.70599,Z 803.39085,A 90,B 0,C -180,S 2,T 35,E1 0,E2 0,E3 0,E4 0,E5 0,E6 0}
   E6POS P2_N_1_Place={X 83.08067,Y 567.70599,Z 653.39085,A 90,B 0,C -180,S 2,T 35,E1 0,E2 0,E3 0,E4 0,E5 0,E6 0}
   E6POS P2_N_2_App1Place={X 658.69065,Y 231.29356,Z 953.39146,A 0,B 0,C -180,S 2,T 35,E1 0,E2 0,E3 0,E4 0,E5 0,E6 0}
   E6POS P2_N_2_App2Place={X 658.69044,Y 231.29349,Z 803.39085,A 0,B 0,C -180,S 2,T 35,E1 0,E2 0,E3 0,E4 0,E5 0,E6 0}
   E6POS P2_N_2_Place={X 658.68978,Y 381.29352,Z 653.39085,A 0,B 0,C 180,S 2,T 35,E1 0,E2 0,E3 0,E4 0,E5 0,E6 0}
   E6POS P2_N_3_App1Place={X 401.08391,Y 1121.71602,Z 953.39146,A 90,B 0,C 180,S 2,T 35,E1 0,E2 0,E3 0,E4 0,E5 0,E6 0}
   E6POS P2_N_3_App2Place={X 401.08405,Y 1121.7159,Z 803.39085,A 90,B 0,C 180,S 2,T 35,E1 0,E2 0,E3 0,E4 0,E5 0,E6 0}
   E6POS P2_N_3_Place={X 301.08415,Y 1071.71593,Z 653.39085,A 90,B 0,C 180,S 2,T 35,E1 0,E2 0,E3 0,E4 0,E5 0,E6 0}
   E6POS P2_N_4_App1Place={X -97.28919,Y 63.29373,Z 953.39146,A 0,B 0,C -180,S 2,T 51,E1 0,E2 0,E3 0,E4 0,E5 0,E6 0}
   E6POS P2_N_4_App2Place={X -97.28973,Y 63.29387,Z 803.39085,A 0,B 0,C 180,S 2,T 51,E1 0,E2 0,E3 0,E4 0,E5 0,E6 0}
   E6POS P2_N_4_Place={X -97.28973,Y 163.29387,Z 653.39085,A 0,B 0,C 180,S 2,T 51,E1 0,E2 0,E3 0,E4 0,E5 0,E6 0}
   E6POS P2_N_5_App1Place={X 687.08177,Y 635.72589,Z 953.39146,A 90,B 0,C 180,S 2,T 35,E1 0,E2 0,E3 0,E4 0,E5 0,E6 0}
   E6POS P2_N_5_App2Place={X 687.08127,Y 635.72551,Z 803.39085,A 90,B 0,C 180,S 2,T 35,E1 0,E2 0,E3 0,E4 0,E5 0,E6 0}
   E6POS P2_N_5_Place={X 587.08127,Y 635.72551,Z 653.39085,A 90,B 0,C 180,S 2,T 35,E1 0,E2 0,E3 0,E4 0,E5 0,E6 0}
   E6POS P2_N_6_App1Place={X 1138.64884,Y 916.0959,Z 953.39146,A -180,B 0,C 180,S 2,T 35,E1 0,E2 0,E3 0,E4 0,E5 0,E6 0}
   E6POS P2_N_6_App2Place={X 1138.6483,Y 916.09602,Z 803.39085,A 180,B 0,C 180,S 2,T 35,E1 0,E2 0,E3 0,E4 0,E5 0,E6 0}
   E6POS P2_N_6_Place={X 1088.6483,Y 816.09602,Z 653.39085,A 180,B 0,C 180,S 2,T 35,E1 0,E2 0,E3 0,E4 0,E5 0,E6 0}
   E6POS P2_N_7_App1Place={X 905.08028,Y 81.72627,Z 953.39146,A 90,B 0,C 180,S 2,T 35,E1 0,E2 0,E3 0,E4 0,E5 0,E6 0}
   E6POS P2_N_7_App2Place={X 905.08036,Y 81.72604,Z 803.39085,A 90,B 0,C 180,S 2,T 51,E1 0,E2 0,E3 0,E4 0,E5 0,E6 0}
   E6POS P2_N_7_Place={X 805.08036,Y 131.72605,Z 653.39085,A 90,B 0,C 180,S 2,T 51,E1 0,E2 0,E3 0,E4 0,E5 0,E6 0}
   E6POS P2_N_8_App1Place={X 1188.64826,Y 1134.09622,Z 953.39146,A -180,B 0,C 180,S 2,T 35,E1 0,E2 0,E3 0,E4 0,E5 0,E6 0}
   E6POS P2_N_8_App2Place={X 1188.64815,Y 1134.09646,Z 803.39085,A -180,B 0,C 180,S 2,T 35,E1 0,E2 0,E3 0,E4 0,E5 0,E6 0}
   E6POS P2_N_8_Place={X 1088.6488,Y 1034.09614,Z 653.39085,A -180,B 0,C 180,S 2,T 35,E1 0,E2 0,E3 0,E4 0,E5 0,E6 0}

   ;ENDFOLD
   ;FOLD  MosaicoO_Pallet2

   E6POS P2_O_1_App1Place={X 935.79484,Y 172.66092,Z 845.88507,A -180,B 0,C 180,S 2,T 35,E1 0,E2 0,E3 0,E4 0,E5 0,E6 0}
   E6POS P2_O_1_App2Place={X 935.79436,Y 172.66159,Z 745.8848,A -180,B 0,C 180,S 2,T 35,E1 0,E2 0,E3 0,E4 0,E5 0,E6 0}
   E6POS P2_O_1_Place={X 935.79476,Y 72.66105,Z 645.88524,A -180,B 0,C 180,S 2,T 51,E1 0,E2 0,E3 0,E4 0,E5 0,E6 0}
   E6POS P2_O_2_App1Place={X 329.01301,Y 456.78538,Z 845.88507,A -180,B 0,C 180,S 2,T 35,E1 0,E2 0,E3 0,E4 0,E5 0,E6 0}
   E6POS P2_O_2_App2Place={X 329.01325,Y 456.7853,Z 745.8848,A -180,B 0,C -180,S 2,T 35,E1 0,E2 0,E3 0,E4 0,E5 0,E6 0}
   E6POS P2_O_2_Place={X 329.01323,Y 356.78607,Z 645.88524,A -180,B 0,C -180,S 2,T 51,E1 0,E2 0,E3 0,E4 0,E5 0,E6 0}
   E6POS P2_O_3_App1Place={X 651.79538,Y 780.66149,Z 845.88507,A -180,B 0,C 180,S 2,T 35,E1 0,E2 0,E3 0,E4 0,E5 0,E6 0}
   E6POS P2_O_3_App2Place={X 651.79565,Y 780.6615,Z 745.8848,A -180,B 0,C -180,S 2,T 35,E1 0,E2 0,E3 0,E4 0,E5 0,E6 0}
   E6POS P2_O_3_Place={X 651.79572,Y 680.66131,Z 645.88524,A -180,B 0,C 180,S 2,T 35,E1 0,E2 0,E3 0,E4 0,E5 0,E6 0}
   E6POS P2_O_4_App1Place={X 45.01175,Y 1064.78615,Z 845.88507,A -180,B 0,C 180,S 2,T 35,E1 0,E2 0,E3 0,E4 0,E5 0,E6 0}
   E6POS P2_O_4_App2Place={X 45.01228,Y 1064.78624,Z 745.8848,A -180,B 0,C 180,S 2,T 35,E1 0,E2 0,E3 0,E4 0,E5 0,E6 0}
   E6POS P2_O_4_Place={X 45.01235,Y 964.78626,Z 645.88524,A -180,B 0,C 180,S 2,T 35,E1 0,E2 0,E3 0,E4 0,E5 0,E6 0}
   E6POS P2_O_5_App1Place={X 170.84994,Y -87.51663,Z 845.88507,A 90,B 0,C 180,S 2,T 51,E1 0,E2 0,E3 0,E4 0,E5 0,E6 0}
   E6POS P2_O_5_App2Place={X 170.85014,Y -87.51635,Z 745.8848,A 90,B 0,C 180,S 2,T 51,E1 0,E2 0,E3 0,E4 0,E5 0,E6 0}
   E6POS P2_O_5_Place={X 270.85006,Y 12.48387,Z 645.88524,A 90,B 0,C 180,S 2,T 51,E1 0,E2 0,E3 0,E4 0,E5 0,E6 0}
   E6POS P2_O_6_App1Place={X 828.97543,Y 1287.26637,Z 845.88507,A -90,B 0,C 180,S 2,T 3,E1 0,E2 0,E3 0,E4 0,E5 0,E6 0}
   E6POS P2_O_6_App2Place={X 828.97552,Y 1287.26658,Z 745.8848,A -90,B 0,C -180,S 2,T 3,E1 0,E2 0,E3 0,E4 0,E5 0,E6 0}
   E6POS P2_O_6_Place={X 714.4457,Y 1187.27407,Z 645.88524,A -90,B 0,C 180,S 2,T 3,E1 0,E2 0,E3 0,E4 0,E5 0,E6 0}
   E6POS P2_O_7_App1Place={X 651.79617,Y 172.66183,Z 845.88507,A -180,B 0,C 180,S 2,T 35,E1 0,E2 0,E3 0,E4 0,E5 0,E6 0}
   E6POS P2_O_7_App2Place={X 651.79644,Y 172.6614,Z 745.8848,A -180,B 0,C -180,S 2,T 35,E1 0,E2 0,E3 0,E4 0,E5 0,E6 0}
   E6POS P2_O_7_Place={X 651.79621,Y 72.66195,Z 645.88524,A -180,B 0,C 180,S 2,T 51,E1 0,E2 0,E3 0,E4 0,E5 0,E6 0}
   E6POS P2_O_8_App1Place={X 45.01334,Y 456.78658,Z 845.88507,A -180,B 0,C 180,S 2,T 35,E1 0,E2 0,E3 0,E4 0,E5 0,E6 0}
   E6POS P2_O_8_App2Place={X 45.01296,Y 456.78657,Z 745.8848,A -180,B 0,C -180,S 2,T 35,E1 0,E2 0,E3 0,E4 0,E5 0,E6 0}
   E6POS P2_O_8_Place={X 45.0129,Y 356.78655,Z 645.88524,A -180,B 0,C -180,S 2,T 35,E1 0,E2 0,E3 0,E4 0,E5 0,E6 0}
   E6POS P2_O_9_App1Place={X 935.79621,Y 780.66179,Z 845.88507,A -180,B 0,C 180,S 2,T 35,E1 0,E2 0,E3 0,E4 0,E5 0,E6 0}
   E6POS P2_O_9_App2Place={X 935.79625,Y 780.66184,Z 745.8848,A -180,B 0,C 180,S 2,T 35,E1 0,E2 0,E3 0,E4 0,E5 0,E6 0}
   E6POS P2_O_9_Place={X 935.79614,Y 680.66184,Z 645.88524,A -180,B 0,C 180,S 2,T 35,E1 0,E2 0,E3 0,E4 0,E5 0,E6 0}
   E6POS P2_O_10_App1Place={X 329.0129,Y 1064.78593,Z 845.88507,A -180,B 0,C 180,S 2,T 35,E1 0,E2 0,E3 0,E4 0,E5 0,E6 0}
   E6POS P2_O_10_App2Place={X 329.0132,Y 1064.78566,Z 745.8848,A -180,B 0,C 180,S 2,T 35,E1 0,E2 0,E3 0,E4 0,E5 0,E6 0}
   E6POS P2_O_10_Place={X 329.01301,Y 964.78561,Z 645.88524,A -180,B 0,C 180,S 2,T 35,E1 0,E2 0,E3 0,E4 0,E5 0,E6 0}
   E6POS P2_O_11_App1Place={X 878.8505,Y -37.51471,Z 845.88507,A 90,B 0,C 180,S 2,T 35,E1 0,E2 0,E3 0,E4 0,E5 0,E6 0}
   E6POS P2_O_11_App2Place={X 878.85073,Y -37.51535,Z 745.8848,A 90,B 0,C 180,S 2,T 35,E1 0,E2 0,E3 0,E4 0,E5 0,E6 0}
   E6POS P2_O_11_Place={X 713.184,Y 15.84173,Z 645.88524,A 90,B 0,C 180,S 2,T 51,E1 0,E2 0,E3 0,E4 0,E5 0,E6 0}
   E6POS P2_O_12_App1Place={X 170.97582,Y 1287.26677,Z 845.88507,A -90,B 0,C 180,S 2,T 35,E1 0,E2 0,E3 0,E4 0,E5 0,E6 0}
   E6POS P2_O_12_App2Place={X 170.97564,Y 1287.26676,Z 745.8848,A -90,B 0,C 180,S 2,T 35,E1 0,E2 0,E3 0,E4 0,E5 0,E6 0}
   E6POS P2_O_12_Place={X 270.97608,Y 1187.26674,Z 645.88524,A -90,B 0,C 180,S 2,T 3,E1 0,E2 0,E3 0,E4 0,E5 0,E6 0}

   ;ENDFOLD
   ;FOLD  MosaicoP2_Pallet2

   E6POS P2_P_1_App1Place={X 617.0748,Y 364.14342,Z 890.16691,A -180,B 0,C 180,S 2,T 35,E1 0,E2 0,E3 0,E4 0,E5 0,E6 0}
   E6POS P2_P_1_App2Place={X 617.07384,Y 364.14354,Z 740.16729,A -180,B 0,C 180,S 2,T 35,E1 0,E2 0,E3 0,E4 0,E5 0,E6 0}
   E6POS P2_P_1_Place={X 616.25932,Y 251.52907,Z 660.09943,A -180,B 0,C 180,S 2,T 51,E1 0,E2 0,E3 0,E4 0,E5 0,E6 0}
   E6POS P2_P_2_App1Place={X 17.29759,Y 778.48787,Z 890.16691,A -180,B 0,C 180,S 2,T 35,E1 0,E2 0,E3 0,E4 0,E5 0,E6 0}
   E6POS P2_P_2_App2Place={X 17.2976,Y 778.48775,Z 740.16729,A -180,B 0,C 180,S 2,T 35,E1 0,E2 0,E3 0,E4 0,E5 0,E6 0}
   E6POS P2_P_2_Place={X 17.29771,Y 665.87327,Z 660.09943,A -180,B 0,C 180,S 2,T 35,E1 0,E2 0,E3 0,E4 0,E5 0,E6 0}
   E6POS P2_P_3_App1Place={X 616.25962,Y 1194.14047,Z 890.16691,A -180,B 0,C 180,S 2,T 35,E1 0,E2 0,E3 0,E4 0,E5 0,E6 0}
   E6POS P2_P_3_App2Place={X 616.25968,Y 1194.1408,Z 740.16729,A -180,B 0,C 180,S 2,T 35,E1 0,E2 0,E3 0,E4 0,E5 0,E6 0}
   E6POS P2_P_3_Place={X 616.25957,Y 1081.52903,Z 660.09943,A -180,B 0,C 180,S 2,T 35,E1 0,E2 0,E3 0,E4 0,E5 0,E6 0}
   E6POS P2_P_4_App1Place={X 1099.0355,Y 595.11551,Z 890.16691,A 90,B 0,C 180,S 2,T 35,E1 0,E2 0,E3 0,E4 0,E5 0,E6 0}
   E6POS P2_P_4_App2Place={X 1099.03552,Y 595.11554,Z 740.16729,A 90,B 0,C 180,S 2,T 35,E1 0,E2 0,E3 0,E4 0,E5 0,E6 0}
   E6POS P2_P_4_Place={X 875.78418,Y 595.11547,Z 660.09943,A 90,B 0,C 180,S 2,T 35,E1 0,E2 0,E3 0,E4 0,E5 0,E6 0}
   E6POS P2_P_5_App1Place={X 986.25995,Y 364.13461,Z 890.16691,A -180,B 0,C -180,S 2,T 35,E1 0,E2 0,E3 0,E4 0,E5 0,E6 0}
   E6POS P2_P_5_App2Place={X 986.25979,Y 364.13425,Z 740.16729,A -180,B 0,C -180,S 2,T 35,E1 0,E2 0,E3 0,E4 0,E5 0,E6 0}
   E6POS P2_P_5_Place={X 986.25884,Y 251.548,Z 660.09943,A -180,B 0,C 180,S 2,T 35,E1 0,E2 0,E3 0,E4 0,E5 0,E6 0}
   E6POS P2_P_6_App1Place={X 387.29628,Y 778.47745,Z 890.16691,A 180,B 0,C 180,S 2,T 35,E1 0,E2 0,E3 0,E4 0,E5 0,E6 0}
   E6POS P2_P_6_App2Place={X 387.29629,Y 778.47753,Z 740.16729,A -180,B 0,C 180,S 2,T 35,E1 0,E2 0,E3 0,E4 0,E5 0,E6 0}
   E6POS P2_P_6_Place={X 387.29686,Y 665.89221,Z 660.09943,A -180,B 0,C 180,S 2,T 35,E1 0,E2 0,E3 0,E4 0,E5 0,E6 0}
   E6POS P2_P_7_App1Place={X 986.2591,Y 1194.13462,Z 890.16691,A -180,B 0,C 180,S 2,T 35,E1 0,E2 0,E3 0,E4 0,E5 0,E6 0}
   E6POS P2_P_7_App2Place={X 986.25917,Y 1194.13486,Z 740.16729,A -180,B 0,C -180,S 2,T 35,E1 0,E2 0,E3 0,E4 0,E5 0,E6 0}
   E6POS P2_P_7_Place={X 986.25895,Y 1081.54783,Z 660.09943,A -180,B 0,C 180,S 2,T 35,E1 0,E2 0,E3 0,E4 0,E5 0,E6 0}
   E6POS P2_P_8_App1Place={X 45.93166,Y 593.04244,Z 890.16691,A -90,B 0,C -180,S 2,T 35,E1 0,E2 0,E3 0,E4 0,E5 0,E6 0}
   E6POS P2_P_8_App2Place={X 45.93167,Y 593.04221,Z 740.16729,A -90,B 0,C 180,S 2,T 35,E1 0,E2 0,E3 0,E4 0,E5 0,E6 0}
   E6POS P2_P_8_Place={X 130.48397,Y 593.04207,Z 660.09943,A -90,B 0,C 180,S 2,T 35,E1 0,E2 0,E3 0,E4 0,E5 0,E6 0}

   ;ENDFOLD
   ;FOLD  MosaicoQ_Pallet2

   E6POS P2_Q_1_App1Place={X 457.55599,Y 375.41531,Z 1111.95686,A -180,B 0,C 180,S 2,T 35,E1 0,E2 0,E3 0,E4 0,E5 0,E6 0}
   E6POS P2_Q_1_App2Place={X 457.55558,Y 375.41581,Z 911.95694,A -180,B 0,C -180,S 2,T 35,E1 0,E2 0,E3 0,E4 0,E5 0,E6 0}
   E6POS P2_Q_1_Place={X 457.5548,Y 275.41596,Z 661.95611,A -180,B 0,C 180,S 2,T 51,E1 0,E2 0,E3 0,E4 0,E5 0,E6 0}
   E6POS P2_Q_2_App1Place={X 558.55551,Y 1099.4166,Z 1111.95686,A -180,B 0,C 180,S 2,T 35,E1 0,E2 0,E3 0,E4 0,E5 0,E6 0}
   E6POS P2_Q_2_App2Place={X 558.55601,Y 1099.41679,Z 911.95694,A -180,B 0,C 180,S 2,T 35,E1 0,E2 0,E3 0,E4 0,E5 0,E6 0}
   E6POS P2_Q_2_Place={X 558.55592,Y 999.41595,Z 661.95611,A -180,B 0,C -180,S 2,T 35,E1 0,E2 0,E3 0,E4 0,E5 0,E6 0}
   E6POS P2_Q_3_App1Place={X 936.32721,Y 1166.50729,Z 1111.95686,A -90,B 0,C 180,S 2,T 3,E1 0,E2 0,E3 0,E4 0,E5 0,E6 0}
   E6POS P2_Q_3_App2Place={X 936.32726,Y 1166.50773,Z 911.95694,A -90,B 0,C -180,S 2,T 3,E1 0,E2 0,E3 0,E4 0,E5 0,E6 0}
   E6POS P2_Q_3_Place={X 836.32776,Y 1066.50753,Z 661.95611,A -90,B 0,C 180,S 2,T 3,E1 0,E2 0,E3 0,E4 0,E5 0,E6 0}
   E6POS P2_Q_4_App1Place={X 40.56894,Y 30.41369,Z 1111.95686,A 90,B 0,C 180,S 2,T 35,E1 0,E2 0,E3 0,E4 0,E5 0,E6 0}
   E6POS P2_Q_4_App2Place={X 40.56901,Y 30.41346,Z 911.95694,A 90,B 0,C 180,S 2,T 51,E1 0,E2 0,E3 0,E4 0,E5 0,E6 0}
   E6POS P2_Q_4_Place={X 140.56858,Y 130.41377,Z 661.95611,A 90,B 0,C 180,S 2,T 51,E1 0,E2 0,E3 0,E4 0,E5 0,E6 0}

   ;ENDFOLD
   ;FOLD  MosaicoR_Pallet2

   E6POS P2_R_1_App1Place={X 899.62721,Y 611.46539,Z 1052.81498,A -90,B 0,C 180,S 2,T 3,E1 0,E2 0,E3 0,E4 0,E5 0,E6 0}
   E6POS P2_R_1_App2Place={X 899.62683,Y 611.4655,Z 852.81474,A -90,B 0,C 180,S 2,T 3,E1 0,E2 0,E3 0,E4 0,E5 0,E6 0}
   E6POS P2_R_1_Place={X 899.62697,Y 561.46554,Z 652.81447,A -90,B 0,C 180,S 2,T 3,E1 0,E2 0,E3 0,E4 0,E5 0,E6 0}
   E6POS P2_R_2_App1Place={X 455.62678,Y 147.46548,Z 1052.81498,A -90,B 0,C 180,S 2,T 3,E1 0,E2 0,E3 0,E4 0,E5 0,E6 0}
   E6POS P2_R_2_App2Place={X 455.62664,Y 147.46525,Z 852.81474,A -90,B 0,C 180,S 2,T 19,E1 0,E2 0,E3 0,E4 0,E5 0,E6 0}
   E6POS P2_R_2_Place={X 555.62602,Y 97.46514,Z 652.81447,A -90,B 0,C 180,S 2,T 19,E1 0,E2 0,E3 0,E4 0,E5 0,E6 0}
   E6POS P2_R_3_App1Place={X 726.31085,Y 877.74519,Z 1052.81498,A -180,B 0,C 180,S 2,T 35,E1 0,E2 0,E3 0,E4 0,E5 0,E6 0}
   E6POS P2_R_3_App2Place={X 726.31138,Y 877.74506,Z 852.81474,A -180,B 0,C 180,S 2,T 35,E1 0,E2 0,E3 0,E4 0,E5 0,E6 0}
   E6POS P2_R_3_Place={X 726.31131,Y 777.74518,Z 652.81447,A -180,B 0,C -180,S 2,T 35,E1 0,E2 0,E3 0,E4 0,E5 0,E6 0}
   E6POS P2_R_4_App1Place={X 38.31125,Y 1109.74485,Z 1052.81498,A -180,B 0,C 180,S 2,T 35,E1 0,E2 0,E3 0,E4 0,E5 0,E6 0}
   E6POS P2_R_4_App2Place={X 38.31117,Y 1109.74517,Z 852.81474,A -180,B 0,C -180,S 2,T 35,E1 0,E2 0,E3 0,E4 0,E5 0,E6 0}
   E6POS P2_R_4_Place={X 38.31156,Y 1009.7447,Z 652.81447,A -180,B 0,C 180,S 2,T 35,E1 0,E2 0,E3 0,E4 0,E5 0,E6 0}
   E6POS P2_R_5_App1Place={X 887.91749,Y 1249.24741,Z 1052.81498,A -90,B 0,C 180,S 2,T 3,E1 0,E2 0,E3 0,E4 0,E5 0,E6 0}
   E6POS P2_R_5_App2Place={X 887.9177,Y 1249.24742,Z 852.81474,A -90,B 0,C 180,S 2,T 3,E1 0,E2 0,E3 0,E4 0,E5 0,E6 0}
   E6POS P2_R_5_Place={X 787.91718,Y 1179.24698,Z 652.81447,A -90,B 0,C 180,S 2,T 3,E1 0,E2 0,E3 0,E4 0,E5 0,E6 0}
   E6POS P2_R_6_App1Place={X 153.87909,Y -80.39772,Z 1052.81498,A 90,B 0,C 180,S 2,T 51,E1 0,E2 0,E3 0,E4 0,E5 0,E6 0}
   E6POS P2_R_6_App2Place={X 153.8784,Y -80.39794,Z 852.81474,A 90,B 0,C 180,S 2,T 51,E1 0,E2 0,E3 0,E4 0,E5 0,E6 0}
   E6POS P2_R_6_Place={X 203.8784,Y 19.60206,Z 652.81447,A 90,B 0,C 180,S 2,T 51,E1 0,E2 0,E3 0,E4 0,E5 0,E6 0}
   E6POS P2_R_7_App1Place={X 899.62807,Y 1307.12163,Z 1052.81498,A -90,B 0,C 180,S 2,T 3,E1 0,E2 0,E3 0,E4 0,E5 0,E6 0}
   E6POS P2_R_7_App2Place={X 899.62822,Y 1307.12121,Z 852.81474,A -90,B 0,C 180,S 2,T 3,E1 0,E2 0,E3 0,E4 0,E5 0,E6 0}
   E6POS P2_R_7_Place={X 899.62822,Y 1257.12121,Z 652.81447,A -90,B 0,C 180,S 2,T 3,E1 0,E2 0,E3 0,E4 0,E5 0,E6 0}
   E6POS P2_R_8_App1Place={X 455.62762,Y 561.12134,Z 1052.81498,A -90,B 0,C 180,S 2,T 3,E1 0,E2 0,E3 0,E4 0,E5 0,E6 0}
   E6POS P2_R_8_App2Place={X 455.62748,Y 561.12122,Z 852.81474,A -90,B 0,C 180,S 2,T 3,E1 0,E2 0,E3 0,E4 0,E5 0,E6 0}
   E6POS P2_R_8_Place={X 555.62748,Y 561.12122,Z 652.81447,A -90,B 0,C 180,S 2,T 3,E1 0,E2 0,E3 0,E4 0,E5 0,E6 0}
   E6POS P2_R_9_App1Place={X 725.42721,Y 321.99995,Z 1052.81498,A -180,B 0,C 180,S 2,T 35,E1 0,E2 0,E3 0,E4 0,E5 0,E6 0}
   E6POS P2_R_9_App2Place={X 725.42713,Y 321.99976,Z 852.81474,A 180,B 0,C 180,S 2,T 35,E1 0,E2 0,E3 0,E4 0,E5 0,E6 0}
   E6POS P2_R_9_Place={X 725.42713,Y 421.99976,Z 652.81447,A 180,B 0,C 180,S 2,T 35,E1 0,E2 0,E3 0,E4 0,E5 0,E6 0}
   E6POS P2_R_10_App1Place={X 37.43578,Y 89.98554,Z 1052.81498,A -180,B 0,C 180,S 2,T 35,E1 0,E2 0,E3 0,E4 0,E5 0,E6 0}
   E6POS P2_R_10_App2Place={X 37.436,Y 89.98561,Z 852.81474,A 180,B 0,C 180,S 2,T 35,E1 0,E2 0,E3 0,E4 0,E5 0,E6 0}
   E6POS P2_R_10_Place={X 37.436,Y 189.98561,Z 652.81447,A 180,B 0,C 180,S 2,T 35,E1 0,E2 0,E3 0,E4 0,E5 0,E6 0}
   E6POS P2_R_11_App1Place={X 157.81229,Y 1230.13243,Z 1052.81498,A -90,B 0,C 180,S 2,T 35,E1 0,E2 0,E3 0,E4 0,E5 0,E6 0}
   E6POS P2_R_11_App2Place={X 157.81214,Y 1230.1328,Z 852.81474,A -90.00001,B 0,C 180,S 2,T 35,E1 0,E2 0,E3 0,E4 0,E5 0,E6 0}
   E6POS P2_R_11_Place={X 207.81214,Y 1180.1328,Z 652.81447,A -90.00001,B 0,C 180,S 2,T 3,E1 0,E2 0,E3 0,E4 0,E5 0,E6 0}
   E6POS P2_R_12_App1Place={X 837.91685,Y -30.40418,Z 1052.81498,A 90,B 0,C 180,S 2,T 35,E1 0,E2 0,E3 0,E4 0,E5 0,E6 0}
   E6POS P2_R_12_App2Place={X 837.91671,Y -30.40437,Z 852.81474,A 90,B 0,C 180,S 2,T 35,E1 0,E2 0,E3 0,E4 0,E5 0,E6 0}
   E6POS P2_R_12_Place={X 787.91779,Y 19.59586,Z 652.81447,A 90,B 0,C 180,S 2,T 35,E1 0,E2 0,E3 0,E4 0,E5 0,E6 0}

   ;ENDFOLD
   ;FOLD  MosaicoS_Pallet2

   E6POS P2_S_1_App1Place={X 741.07837,Y 636.24248,Z 1090.17086,A -89.99997,B 0,C -180,S 2,T 3,E1 0,E2 0,E3 0,E4 0,E5 0,E6 0}
   E6POS P2_S_1_App2Place={X 741.07843,Y 636.24271,Z 890.17129,A -89.99997,B 0,C 180,S 2,T 3,E1 0,E2 0,E3 0,E4 0,E5 0,E6 0}
   E6POS P2_S_1_Place={X 910.50314,Y 581.88157,Z 662.05452,A -89.99997,B 0,C 180,S 2,T 3,E1 0,E2 0,E3 0,E4 0,E5 0,E6 0}
   E6POS P2_S_2_App1Place={X 418.07874,Y 636.74259,Z 1090.17086,A -90,B 0,C 180,S 2,T 3,E1 0,E2 0,E3 0,E4 0,E5 0,E6 0}
   E6POS P2_S_2_App2Place={X 418.07876,Y 636.74273,Z 890.17129,A -90,B 0,C 180,S 2,T 3,E1 0,E2 0,E3 0,E4 0,E5 0,E6 0}
   E6POS P2_S_2_Place={X 587.50395,Y 582.38133,Z 662.05452,A -90,B 0,C 180,S 2,T 3,E1 0,E2 0,E3 0,E4 0,E5 0,E6 0}
   E6POS P2_S_3_App1Place={X 163.70727,Y 108.33204,Z 1090.17086,A -90,B 0,C 180,S 2,T 35,E1 0,E2 0,E3 0,E4 0,E5 0,E6 0}
   E6POS P2_S_3_App2Place={X 163.70752,Y 108.33171,Z 890.17129,A -90,B 0,C -180,S 2,T 51,E1 0,E2 0,E3 0,E4 0,E5 0,E6 0}
   E6POS P2_S_3_Place={X 263.70752,Y 108.33171,Z 662.05452,A -90,B 0,C -180,S 2,T 19,E1 0,E2 0,E3 0,E4 0,E5 0,E6 0}
   E6POS P2_S_4_App1Place={X 548.9828,Y 698.88733,Z 1090.17086,A 180,B 0,C 180,S 2,T 35,E1 0,E2 0,E3 0,E4 0,E5 0,E6 0}
   E6POS P2_S_4_App2Place={X 548.98283,Y 698.88748,Z 890.17129,A -180,B 0,C 180,S 2,T 35,E1 0,E2 0,E3 0,E4 0,E5 0,E6 0}
   E6POS P2_S_4_Place={X 548.98171,Y 596.91087,Z 662.05452,A -180,B 0,C 180,S 2,T 35,E1 0,E2 0,E3 0,E4 0,E5 0,E6 0}
   E6POS P2_S_5_App1Place={X 548.98204,Y 1001.8871,Z 1090.17086,A 180,B 0,C 180,S 2,T 35,E1 0,E2 0,E3 0,E4 0,E5 0,E6 0}
   E6POS P2_S_5_App2Place={X 548.98207,Y 1001.88729,Z 890.17129,A -180,B 0,C 180,S 2,T 35,E1 0,E2 0,E3 0,E4 0,E5 0,E6 0}
   E6POS P2_S_5_Place={X 548.98218,Y 899.91031,Z 662.05452,A -180,B 0,C -180,S 2,T 35,E1 0,E2 0,E3 0,E4 0,E5 0,E6 0}
   E6POS P2_S_6_App1Place={X 212.99282,Y 614.54248,Z 1090.17086,A 90,B 0,C 180,S 2,T 35,E1 0,E2 0,E3 0,E4 0,E5 0,E6 0}
   E6POS P2_S_6_App2Place={X 212.99282,Y 614.54256,Z 890.17129,A 90,B 0,C 180,S 2,T 35,E1 0,E2 0,E3 0,E4 0,E5 0,E6 0}
   E6POS P2_S_6_Place={X 88.77457,Y 614.54268,Z 662.05452,A 90,B 0,C 180,S 2,T 35,E1 0,E2 0,E3 0,E4 0,E5 0,E6 0}
   E6POS P2_S_7_App1Place={X 535.99307,Y 614.14253,Z 1090.17086,A 90,B 0,C -180,S 2,T 35,E1 0,E2 0,E3 0,E4 0,E5 0,E6 0}
   E6POS P2_S_7_App2Place={X 535.99309,Y 614.14264,Z 890.17129,A 90,B 0,C 180,S 2,T 35,E1 0,E2 0,E3 0,E4 0,E5 0,E6 0}
   E6POS P2_S_7_Place={X 411.77415,Y 614.14281,Z 662.05452,A 90,B 0,C 180,S 2,T 35,E1 0,E2 0,E3 0,E4 0,E5 0,E6 0}
   E6POS P2_S_8_App1Place={X 834.59206,Y 1088.58923,Z 1090.17086,A 90,B 0,C 180,S 2,T 35,E1 0,E2 0,E3 0,E4 0,E5 0,E6 0}
   E6POS P2_S_8_App2Place={X 834.59246,Y 1088.58903,Z 890.17129,A 90,B 0,C 180,S 2,T 35,E1 0,E2 0,E3 0,E4 0,E5 0,E6 0}
   E6POS P2_S_8_Place={X 734.59246,Y 1088.58903,Z 662.05452,A 90,B 0,C 180,S 2,T 35,E1 0,E2 0,E3 0,E4 0,E5 0,E6 0}
   E6POS P2_S_9_App1Place={X 449.28082,Y 499.5508,Z 1090.17086,A 0,B 0,C -180,S 2,T 3,E1 0,E2 0,E3 0,E4 0,E5 0,E6 0}
   E6POS P2_S_9_App2Place={X 449.28084,Y 499.55095,Z 890.17129,A 0,B 0,C -180,S 2,T 3,E1 0,E2 0,E3 0,E4 0,E5 0,E6 0}
   E6POS P2_S_9_Place={X 449.28092,Y 599.55096,Z 662.05452,A 0,B 0,C 180,S 2,T 3,E1 0,E2 0,E3 0,E4 0,E5 0,E6 0}
   E6POS P2_S_10_App1Place={X 449.28449,Y 196.54354,Z 1090.17086,A 0,B 0,C -180,S 2,T 3,E1 0,E2 0,E3 0,E4 0,E5 0,E6 0}
   E6POS P2_S_10_App2Place={X 449.28452,Y 196.54376,Z 890.17129,A 0,B 0,C -180,S 2,T 3,E1 0,E2 0,E3 0,E4 0,E5 0,E6 0}
   E6POS P2_S_10_Place={X 449.285,Y 296.54355,Z 662.05452,A 0,B 0,C 180,S 2,T 3,E1 0,E2 0,E3 0,E4 0,E5 0,E6 0}

   ;ENDFOLD
   ;FOLD  MosaicoT_Pallet2

   E6POS P2_T_1_App1Place={X 519.6645,Y 1058.50264,Z 970.17241,A -180,B 0,C 180,S 2,T 35,E1 0,E2 0,E3 0,E4 0,E5 0,E6 0}
   E6POS P2_T_1_App2Place={X 519.66406,Y 1058.50233,Z 820.17205,A 180,B 0,C 180,S 2,T 35,E1 0,E2 0,E3 0,E4 0,E5 0,E6 0}
   E6POS P2_T_1_Place={X 519.66406,Y 1108.50233,Z 670.17205,A 180,B 0,C 180,S 2,T 35,E1 0,E2 0,E3 0,E4 0,E5 0,E6 0}
   E6POS P2_T_2_App1Place={X 519.66406,Y 1108.50233,Z 970.17241,A 180,B 0,C 180,S 2,T 35,E1 0,E2 0,E3 0,E4 0,E5 0,E6 0}
   E6POS P2_T_2_App2Place={X 550.66406,Y 1108.50233,Z 820.17205,A 180,B 0,C 180,S 2,T 35,E1 0,E2 0,E3 0,E4 0,E5 0,E6 0}
   E6POS P2_T_2_Place={X 550.66406,Y 1108.50233,Z 670.17205,A 180,B 0,C 180,S 2,T 35,E1 0,E2 0,E3 0,E4 0,E5 0,E6 0}
   E6POS P2_T_3_App1Place={X 550.66406,Y 1108.50233,Z 970.17241,A 180,B 0,C 180,S 2,T 35,E1 0,E2 0,E3 0,E4 0,E5 0,E6 0}
   E6POS P2_T_3_App2Place={X 581.66406,Y 1108.50233,Z 820.17205,A 180,B 0,C 180,S 2,T 35,E1 0,E2 0,E3 0,E4 0,E5 0,E6 0}
   E6POS P2_T_3_Place={X 581.66406,Y 1108.50233,Z 670.17205,A 180,B 0,C 180,S 2,T 35,E1 0,E2 0,E3 0,E4 0,E5 0,E6 0}
   E6POS P2_T_4_App1Place={X 519.68064,Y 803.68323,Z 970.17241,A -180,B 0,C 180,S 2,T 35,E1 0,E2 0,E3 0,E4 0,E5 0,E6 0}
   E6POS P2_T_4_App2Place={X 519.68029,Y 803.68307,Z 820.17205,A 180,B 0,C 180,S 2,T 35,E1 0,E2 0,E3 0,E4 0,E5 0,E6 0}
   E6POS P2_T_4_Place={X 519.68029,Y 903.68307,Z 670.17205,A 180,B 0,C -180,S 2,T 35,E1 0,E2 0,E3 0,E4 0,E5 0,E6 0}
   E6POS P2_T_5_App1Place={X 519.67999,Y 490.68329,Z 970.17241,A -180,B 0,C 180,S 2,T 35,E1 0,E2 0,E3 0,E4 0,E5 0,E6 0}
   E6POS P2_T_5_App2Place={X 519.68029,Y 490.68307,Z 820.17205,A 180,B 0,C 180,S 2,T 35,E1 0,E2 0,E3 0,E4 0,E5 0,E6 0}
   E6POS P2_T_5_Place={X 519.68031,Y 590.68319,Z 670.17205,A 180,B 0,C 180,S 2,T 35,E1 0,E2 0,E3 0,E4 0,E5 0,E6 0}
   E6POS P2_T_6_App1Place={X 519.68061,Y 177.68258,Z 970.17241,A -180,B 0,C 180,S 2,T 35,E1 0,E2 0,E3 0,E4 0,E5 0,E6 0}
   E6POS P2_T_6_App2Place={X 519.68029,Y 177.68307,Z 820.17205,A 180,B 0,C 180,S 2,T 51,E1 0,E2 0,E3 0,E4 0,E5 0,E6 0}
   E6POS P2_T_6_Place={X 519.68029,Y 277.68303,Z 670.17205,A 180,B 0,C 180,S 2,T 51,E1 0,E2 0,E3 0,E4 0,E5 0,E6 0}
   E6POS P2_T_7_App1Place={X 519.68061,Y 1003.68258,Z 970.17241,A -180,B 0,C 180,S 2,T 35,E1 0,E2 0,E3 0,E4 0,E5 0,E6 0}
   E6POS P2_T_7_App2Place={X 519.68029,Y 1003.68307,Z 820.17205,A 180,B 0,C 180,S 2,T 35,E1 0,E2 0,E3 0,E4 0,E5 0,E6 0}
   E6POS P2_T_7_Place={X 519.68029,Y 1103.68303,Z 670.17205,A 180,B 0,C 180,S 2,T 35,E1 0,E2 0,E3 0,E4 0,E5 0,E6 0}
   E6POS P2_T_8_App1Place={X 519.68061,Y 690.68258,Z 970.17241,A -180,B 0,C 180,S 2,T 35,E1 0,E2 0,E3 0,E4 0,E5 0,E6 0}
   E6POS P2_T_8_App2Place={X 519.68029,Y 690.68307,Z 820.17205,A 180,B 0,C 180,S 2,T 35,E1 0,E2 0,E3 0,E4 0,E5 0,E6 0}
   E6POS P2_T_8_Place={X 519.68029,Y 790.68303,Z 670.17205,A 180,B 0,C 180,S 2,T 35,E1 0,E2 0,E3 0,E4 0,E5 0,E6 0}
   E6POS P2_T_9_App1Place={X 519.68061,Y 377.68258,Z 970.17241,A -180,B 0,C 180,S 2,T 35,E1 0,E2 0,E3 0,E4 0,E5 0,E6 0}
   E6POS P2_T_9_App2Place={X 519.68029,Y 377.68307,Z 820.17205,A 180,B 0,C 180,S 2,T 35,E1 0,E2 0,E3 0,E4 0,E5 0,E6 0}
   E6POS P2_T_9_Place={X 519.68029,Y 477.68303,Z 670.17205,A 180,B 0,C 180,S 2,T 35,E1 0,E2 0,E3 0,E4 0,E5 0,E6 0}
   E6POS P2_T_10_App1Place={X 519.6645,Y 119.50264,Z 970.17241,A -180,B 0,C 180,S 2,T 35,E1 0,E2 0,E3 0,E4 0,E5 0,E6 0}
   E6POS P2_T_10_App2Place={X 519.66406,Y 119.50233,Z 820.17205,A 180,B 0,C 180,S 2,T 35,E1 0,E2 0,E3 0,E4 0,E5 0,E6 0}
   E6POS P2_T_10_Place={X 519.66406,Y 169.50233,Z 670.17205,A 180,B 0,C 180,S 2,T 35,E1 0,E2 0,E3 0,E4 0,E5 0,E6 0}
   E6POS P2_T_11_App1Place={X 519.66406,Y 169.50233,Z 970.17241,A 180,B 0,C 180,S 2,T 35,E1 0,E2 0,E3 0,E4 0,E5 0,E6 0}
   E6POS P2_T_11_App2Place={X 550.66406,Y 169.50233,Z 820.17205,A 180,B 0,C 180,S 2,T 35,E1 0,E2 0,E3 0,E4 0,E5 0,E6 0}
   E6POS P2_T_11_Place={X 550.66406,Y 169.50233,Z 670.17205,A 180,B 0,C 180,S 2,T 35,E1 0,E2 0,E3 0,E4 0,E5 0,E6 0}
   E6POS P2_T_12_App1Place={X 550.66406,Y 169.50233,Z 970.17241,A 180,B 0,C 180,S 2,T 35,E1 0,E2 0,E3 0,E4 0,E5 0,E6 0}
   E6POS P2_T_12_App2Place={X 581.66406,Y 169.50233,Z 820.17205,A 180,B 0,C 180,S 2,T 35,E1 0,E2 0,E3 0,E4 0,E5 0,E6 0}
   E6POS P2_T_12_Place={X 581.66406,Y 169.50233,Z 670.17205,A 180,B 0,C 180,S 2,T 35,E1 0,E2 0,E3 0,E4 0,E5 0,E6 0}

   ;ENDFOLD

   ;ENDFOLD
ENDDAT
